Staubli VAL3: isAtPoint.pgx

program isAtPoint(num x_nIndex, bool& x_bInside[])
  local point l_pHere
  local tool l_tTool
  local num l_nDistance
  local point l_pPoint[2]
  local num l_nIndexTool
  local TrajectoryItem l_tTrajItem
begin
  // reset the bool
  x_bInside=false
  // get the tcp
  call trajType:getTool(l_nIndexTool)
  call saveData:getTool(l_tTool,l_nIndexTool)
  // get the mdesc
  call trajType:getTrajItem(l_tTrajItem,x_nIndex)
  // get the acutal point
  l_pHere=here(l_tTool,world)
  // look if the robot is inside the blend area
  call trajType:getPoint(l_pPoint,false,x_nIndex)
  // check the radius
  if distance(position(l_pPoint,world),l_pHere.trsf)<=max(l_nDistance,nRoundStepping)
    x_bInside=true
  endIf
end
